// TIA Portal V20 export
TYPE "LER_typeVisionResultDataReelCut"
// stored: Access Published
   STRUCT
      tabLength_JudgementResult : Real;   // Tab length_Judgement Result (0:NONE,1:OK,2:NG)
      tabHeight_JudgementResult : Real;   // Tab Height_Judgement Result (0:NONE,1:OK,2:NG)
      electrodeLength_JudgementResult : Real;   // Electrode length_Judgement Result (0:NONE,1:OK,2:NG)
      electrodeHeight_JudgementResult : Real;   // Electrode height_Judgement Result (0:NONE,1:OK,2:NG)
      gapToTabLeftEdge_JudgementResult : Real;   // Gap ↔ Tab left Edge_Judgement Result (0:NONE,1:OK,2:NG)
      gapToTabRightEdge_JudgementResult : Real;   // Gap ↔ Tab right Edge_Judgement Result (0:NONE,1:OK,2:NG)
      totalElectrodeHeightY_JudgementResult : Real;   // Height (y) of total electrode (ini. Tab)_Judgement Result (0:NONE,1:OK,2:NG)
      ceramicCoatingHeight_JudgementResult : Real;   // Height of Ceramic Coating_Judgement Result (0:NONE,1:OK,2:NG)(Cathode Only)
      radiusMeasurement_JudgementResult : Real;   // Radi Measurement_Judgement Result (0:NONE,1:OK,2:NG)
      spare_1 : Real;
      spare_2 : Real;
      spare_3 : Real;
      spare_4 : Real;
      spare_5 : Real;
      spare_6 : Real;
      spare_7 : Real;
      spare_8 : Real;
      spare_9 : Real;
      spare_10 : Real;
      spare_11 : Real;
      TabLength_Reply : Real;   // Tab length_Reply [mm](1/1000)
      TabLength_UpperRange : Real;   // Tab length_Upper Range Reply [mm](1/1000)
      TabLength_LowerRange : Real;   // Tab length_Lower Range Reply [mm](1/1000)
      TabHeight_Reply : Real;   // Tab Height Reply [mm](1/1000)
      TabHeight_UpperRange : Real;   // Tab Height(1/1000) Upper Range Reply [mm](1/1000)
      TabHeight_LowerRange : Real;   // Tab Height(1/1000) Lower Range Reply [mm](1/1000)
      ElectrodeLength_Reply : Real;   // Electrode length_Reply [mm](1/1000)
      ElectrodeLength_UpperRange : Real;   // Electrode length_Upper Range Reply [mm](1/1000)
      ElectrodeLength_LowerRange : Real;   // Electrode length_Lower Range Reply [mm](1/1000)
      ElectrodeHeight_Reply : Real;   // Electrode height_Reply [mm](1/1000)
      ElectrodeHeight_UpperRange : Real;   // Electrode height(1/1000) Upper Range Reply [mm](1/1000)
      ElectrodeHeight_LowerRange : Real;   // Electrode height(1/1000) Lower Range Reply [mm](1/1000)
      Gap_TabLeftEdge_Reply : Real;   // Gap ↔ Tab Left Edge_Reply [mm](1/1000)
      Gap_TabLeftEdge_UpperRange : Real;   // Gap ↔ Tab Left Edge_Upper Range Reply [mm](1/1000)
      Gap_TabLeftEdge_LowerRange : Real;   // Gap ↔ Tab Left Edge_Lower Range Reply [mm](1/1000)
      Gap_TabRightEdge_Reply : Real;   // Gap ↔ Tab right Edge_Reply [mm](1/1000)
      Gap_TabRightEdge_UpperRange : Real;   // Gap ↔ Tab right Edge_Upper Range Reply [mm](1/1000)
      Gap_TabRightEdge_LowerRange : Real;   // Gap ↔ Tab right Edge_Lower Range Reply [mm](1/1000)
      TotalElectrodeHeight_Reply : Real;   // Height (y) of total electrode (ini. Tab)_Reply [mm](1/1000)
      TotalElectrodeHeight_UpperRange : Real;   // Height (y) of total electrode (ini. Tab)_Upper Range Reply [mm](1/1000)
      TotalElectrodeHeight_LowerRange : Real;   // Height (y) of total electrode (ini. Tab)_Lower Range Reply [mm](1/1000)
      CeramicCoatingHeight_Reply : Real;   // Height of Ceramic Coatingy [mm](1/1000) (Cathode Only)
      CeramicCoatingHeight_UpperRange : Real;   // Height of Ceramic Coating_Upper Range Reply [mm](1/1000) (Cathode Only)
      CeramicCoatingHeight_LowerRange : Real;   // Height of Ceramic Coating_Lower Range Reply [mm](1/1000) (Cathode Only)
      RadiusMeasurement_Reply : Real;   // Radi Measurement_Reply [mm](1/1000)
      RadiusMeasurement_UpperRange : Real;   // Radi Measurement_Upper Range Reply [mm](1/1000)
      RadiusMeasurement_LowerRange : Real;   // Radi Measurement_Lower Range Reply [mm](1/1000)
   END_STRUCT;
END_TYPE
